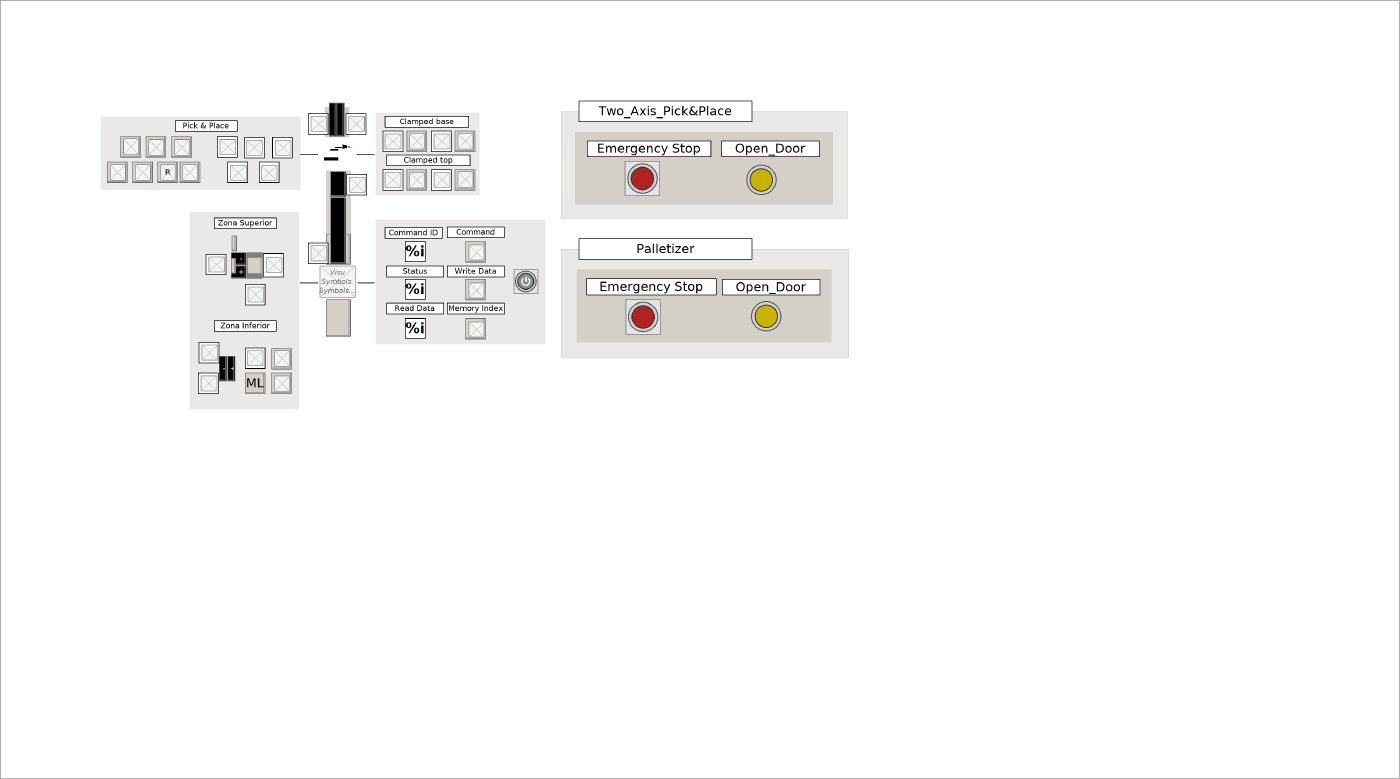
VISUALIZATION Linea_Produccion_Azul_2  // 2001x1114
    Rectangle (1846,508 153x409), angle 90
    Rectangle (827,144 248x30), "Two_Axis_Pick&Place"
    Rectangle (1855,498 103x368), angle 90
    PushSwitch (893,230 50x50), variable: GVL.Emergency_Stop_3, behaviour: TOGGLE, style: Switch-PushSwitch-Red
    Rectangle (839,201 177x23), "Emergency Stop"
    Lamp1 (1063,232 50x50), variable: NOT GVL.Safety_Door_1 OR NOT GVL.Safety_Door_2, style: Lamp-Lamp1-Yellow
    Rectangle (1031,201 140x23), "Open_Door"
    Rectangle (1846,703 155x411), angle 90
    Rectangle (827,341 248x30), "Palletizer"
    Rectangle (1614,447 104x364), angle 90
    PushSwitch (894,428 50x50), behaviour: TOGGLE, style: Switch-PushSwitch-Red
    Rectangle (838,398 186x24), "Emergency Stop"
    Lamp1 (1070,427 50x50), variable: NOT GVL.Safety_Door_3 OR NOT GVL.Safety_Door_4, style: Lamp-Lamp1-Yellow
    Rectangle (1032,399 140x23), "Open_Door"
    InvisibleInput (880,700 18x108)
    InvisibleInput (1316,220 49x41)
    Rectangle (1327,891 282x156), angle 90
    Rectangle (1569,733 118x148), angle 90
    Rectangle (1340,766 104x285), angle 90
    Button (466,334 35x44), colour toggle: GVL.Roller_Conveyor_2m_1, pressed state: GVL.Roller_Conveyor_2m_1
        OnMouseClick: toggle GVL.Roller_Conveyor_2m_1
    Rectangle (461,157 43x35), angle 90
    Group (456,196 53x49)
        InvisibleInput (0,0 53x49)
        RoundedRectangle (7,29 20x4), angle 107
        RoundedRectangle (16,17 11x2), angle 107
        RoundedRectangle (23,14 11x1), angle 180
        Polygon (33,10) (40,12) (40,14) (40,15) (33,17)
        Polygon (47,14) (47,14) (41,14) (41,14) (41,13)
    Rectangle (440,271 89x35), angle 90
    Group (455,378 55x50)
        InvisibleInput (0,0 55x50)
        Image (2,2 51x45), image: VisuSymbols.Symbols.Box
    Line (429,220) (454,220)
    Line (429,404) (454,404)
    Line (511,404) (535,404)
    Button (470,147 11x48), colour toggle: GVL.Belt_Conveyor_4m_6, pressed state: GVL.Belt_Conveyor_4m_6
        OnMouseClick: toggle GVL.Belt_Conveyor_4m_6
    Button (481,147 11x48), colour toggle: GVL.Belt_Conveyor_4m_7, pressed state: GVL.Belt_Conveyor_4m_7
        OnMouseClick: toggle GVL.Belt_Conveyor_4m_7
    Button (472,245 22x36), colour toggle: GVL.Belt_Conveyor_2m_15, pressed state: GVL.Belt_Conveyor_2m_15
        OnMouseClick: toggle GVL.Belt_Conveyor_2m_15
    Button (472,282 22x95), colour toggle: GVL.Belt_Conveyor_Inclined_1, pressed state: GVL.Belt_Conveyor_Inclined_1
        OnMouseClick: toggle GVL.Belt_Conveyor_Inclined_1
    Button (466,428 35x53), colour toggle: GVL.Roller_Conveyor_2m_2, pressed state: GVL.Roller_Conveyor_2m_2
        OnMouseClick: toggle GVL.Roller_Conveyor_2m_2
    Group (440,162 29x30), colour toggle: GVL.Diffuse_Sensor_12
        RoundedRectangle (0,0 29x30), colour toggle: GVL.Diffuse_Sensor_4
        Image (4,4 23x22), image: VisuSymbols.Symbols.RSS1
    Group (494,162 29x30), colour toggle: GVL.Diffuse_Sensor_13
        RoundedRectangle (0,0 29x30), colour toggle: GVL.Diffuse_Sensor_4
        Image (4,4 23x22), image: VisuSymbols.Symbols.RSS1
    Group (495,249 29x30), colour toggle: GVL.Diffuse_Sensor_14
        RoundedRectangle (0,0 29x30), colour toggle: GVL.Diffuse_Sensor_4
        Image (4,4 23x22), image: VisuSymbols.Symbols.RSS1
    Group (440,347 29x30), colour toggle: GVL.Diffuse_Sensor_22
        RoundedRectangle (0,0 29x30), colour toggle: GVL.Diffuse_Sensor_4
        Image (4,4 23x22), image: VisuSymbols.Symbols.RSS1
    Group (310,195 29x30), colour toggle: GVL.Two_Axis_Pick_Place_1_Detected
        RoundedRectangle (0,0 29x30), colour toggle: GVL.Two_Axis_Pick_Place_1_Detected
        Image (4,4 23x22), image: VisuSymbols.Symbols.RSS1
    Group (349,196 29x30), colour toggle: GVL.Two_Axis_Pick_Place_1_MovingX
        RoundedRectangle (0,0 29x30), colour toggle: GVL.Diffuse_Sensor_4
        Image (3,4 23x22), image: VisuSymbols.Symbols.DoubleArrow3
    Group (325,231 29x30), "G", colour toggle: GVL.Two_Axis_Pick_Place_1_Gripper_Rotating
        RoundedRectangle (0,0 29x30), colour toggle: GVL.Diffuse_Sensor_4
        Image (4,5 23x22), image: VisuSymbols.Symbols.ArrowRoundRightDown
    Group (389,196 29x30), colour toggle: GVL.Two_Axis_Pick_Place_1_MovingZ
        RoundedRectangle (0,0 29x30), colour toggle: GVL.Diffuse_Sensor_4
        Image (4,4 23x22), image: VisuSymbols.Symbols.DoubleArrow4
    Group (370,231 29x30), "R", colour toggle: GVL.Two_Axis_Pick_Place_1_Rotating
        RoundedRectangle (0,0 29x30), colour toggle: GVL.Diffuse_Sensor_4
        Image (3,5 23x22), image: VisuSymbols.Symbols.ArrowHalfLeftUp
    Rectangle (250,172 89x16), "Pick & Place"
    Group (547,187 29x30), colour toggle: NOT GVL.Right_Positioner_1_Clamped
        RoundedRectangle (0,0 29x30), colour toggle: GVL.Diffuse_Sensor_4
        Image (3,4 23x22), image: VisuSymbols.Symbols.DoubleArrow3
    Group (616,187 29x30), colour toggle: GVL.Right_Positioner_1_Limit
        RoundedRectangle (0,0 29x30), colour toggle: GVL.Diffuse_Sensor_4
        Image (4,4 23x22), image: VisuSymbols.Symbols.DoubleArrow4
    Rectangle (550,166 120x16), "Clamped base"
    Group (547,242 29x30), colour toggle: NOT GVL.Right_Positioner_2_Clamped
        RoundedRectangle (0,0 29x30), colour toggle: GVL.Diffuse_Sensor_4
        Image (3,4 23x22), image: VisuSymbols.Symbols.DoubleArrow3
    Group (616,242 29x30), colour toggle: GVL.Right_Positioner_2_Limit
        RoundedRectangle (0,0 29x30), colour toggle: GVL.Diffuse_Sensor_4
        Image (4,4 23x22), image: VisuSymbols.Symbols.DoubleArrow4
    Rectangle (552,221 120x16), "Clamped top"
    Line (510,220) (535,220)
    Button (330,361 22x18), "-", colour toggle: GVL.Palletizer_1_Belt_menos, pressed state: GVL.Palletizer_1_Belt_menos
        OnMouseClick: toggle GVL.Palletizer_1_Belt_menos
    Button (331,337 7x22), colour toggle: GVL.Palletizer_1_Turn, pressed state: GVL.Palletizer_1_Turn
        OnMouseClick: toggle GVL.Palletizer_1_Turn
    Button (353,361 22x36), colour toggle: GVL.Palletizer_1_Open_Plate, pressed state: GVL.Palletizer_1_Open_Plate
        OnMouseClick: toggle GVL.Palletizer_1_Open_Plate
    Button (353,391 22x7), colour toggle: GVL.Palletizer_1_Clamb, pressed state: GVL.Palletizer_1_Clamb
        OnMouseClick: toggle GVL.Palletizer_1_Clamb
    Group (350,406 29x30), colour toggle: GVL.Palletizer_1_Clamped
        RoundedRectangle (0,0 29x30), colour toggle: GVL.Diffuse_Sensor_4
        Image (4,4 23x22), image: VisuSymbols.Symbols.DoubleArrow4
    Group (376,362 29x34), colour toggle: GVL.Palletizer_1_Plate_Limit
        RoundedRectangle (0,0 29x34), colour toggle: GVL.Diffuse_Sensor_4
        Image (4,6 23x22), angle 45, image: VisuSymbols.Symbols.DoubleArrow1
    Button (330,380 22x18), "+", colour toggle: GVL.Palletizer_1_Belt_mas, pressed state: GVL.Palletizer_1_Belt_mas
        OnMouseClick: toggle GVL.Palletizer_1_Belt_mas
    Button (330,369 7x22), colour toggle: GVL.Palletizer_1_Push, pressed state: GVL.Palletizer_1_Push
        OnMouseClick: toggle GVL.Palletizer_1_Push
    Button (353,361 22x7), colour toggle: GVL.Palletizer_1_Clamb, pressed state: GVL.Palletizer_1_Clamb
        OnMouseClick: toggle GVL.Palletizer_1_Clamb
    Group (294,363 29x30), colour toggle: GVL.Palletizer_1_Pusher_Limit
        RoundedRectangle (0,0 29x30), colour toggle: GVL.Diffuse_Sensor_4
        Image (4,4 23x22), image: VisuSymbols.Symbols.ArrowBoldRight
    Button (325,509 11x36), "+", colour toggle: GVL.Palletizer_1_Chain_mas, pressed state: GVL.Palletizer_1_Belt_mas
        OnMouseClick: toggle GVL.Palletizer_1_Chain_mas
    Button (313,509 11x36), "-", colour toggle: GVL.Palletizer_1_Chain_menos, pressed state: GVL.Palletizer_1_Belt_menos
        OnMouseClick: toggle GVL.Palletizer_1_Chain_menos
    Group (284,489 29x30), colour toggle: GVL.Palletizer_1_Elevator_Back_Limit
        RoundedRectangle (0,0 29x30), colour toggle: GVL.Two_Axis_Pick_Place_1_Detected
        Image (4,4 23x22), image: VisuSymbols.Symbols.RSS1
    Group (283,533 29x30), colour toggle: GVL.Palletizer_1_Elevator_Front_Limit
        RoundedRectangle (0,0 29x30), colour toggle: GVL.Two_Axis_Pick_Place_1_Detected
        Image (4,4 23x22), image: VisuSymbols.Symbols.RSS1
    Group (350,497 29x30), colour toggle: GVL.Palletizer_1_Elevator_Moving
        RoundedRectangle (0,0 29x30), colour toggle: GVL.Diffuse_Sensor_4
        Image (3,4 23x22), image: VisuSymbols.Symbols.Wheel
    Button (350,533 29x30), "ML", colour toggle: GVL.Palletizer_1_Elevator_Move_Limit, pressed state: GVL.Palletizer_1_Open_Plate
        OnMouseClick: toggle GVL.Palletizer_1_Elevator_Move_Limit
    Group (388,498 29x30), colour toggle: GVL.Palletizer_1_Elevator_mas
        OnMouseClick: toggle GVL.Palletizer_1_Elevator_mas
        Button (0,0 29x30)
        Image (4,3 22x23), image: VisuSymbols.Symbols.ArrowBoldUp
    Group (388,533 29x30), colour toggle: GVL.Palletizer_1_Elevator_menos
        OnMouseClick: toggle GVL.Palletizer_1_Elevator_menos
        Button (0,0 29x30)
        Image (4,4 22x23), image: VisuSymbols.Symbols.ArrowBoldDown
    Rectangle (306,311 89x16), "Zona Superior"
    Rectangle (306,458 89x16), "Zona Inferior"
    Group (208,195 29x30), colour toggle: GVL.Two_Axis_Pick_Place_1X
        OnMouseClick: toggle GVL.Two_Axis_Pick_Place_1X
        Button (0,0 29x30)
        Image (4,4 22x23), image: VisuSymbols.Symbols.ArrowBoldRight
    Group (172,195 29x30), colour toggle: GVL.Two_Axis_Pick_Place_1_Grab
        OnMouseClick: toggle GVL.Two_Axis_Pick_Place_1_Grab
        Button (0,0 29x30)
        Image (4,3 22x23), image: VisuSymbols.Symbols.Download
    Group (257,231 29x30), colour toggle: GVL.Two_Axis_Pick_Place_1_Rotate_CCW
        OnMouseClick: toggle GVL.Two_Axis_Pick_Place_1_Rotate_CCW
        Button (0,0 29x30)
        Image (3,4 22x23), image: VisuSymbols.Symbols.ArrowHalfLeftUp
    Group (189,231 29x30), colour toggle: GVL.Two_Axis_Pick_Place_1_Gripper_CW
        OnMouseClick: toggle GVL.Two_Axis_Pick_Place_1_Gripper_CW
        Button (0,0 29x30)
        Image (4,4 22x23), image: VisuSymbols.Symbols.ArrowRoundRightDown
    Group (153,231 29x30), colour toggle: GVL.Two_Axis_Pick_Place_1_Gripper_CCW
        OnMouseClick: toggle GVL.Two_Axis_Pick_Place_1_Gripper_CCW
        Button (0,0 29x30)
        Image (4,4 22x23), image: VisuSymbols.Symbols.ArrowRoundLeftBottom
    Group (225,231 29x30), colour toggle: GVL.Two_Axis_Pick_Place_1_Rotare_CW
        OnMouseClick: toggle GVL.Two_Axis_Pick_Place_1_Rotare_CW
        Button (0,0 29x30)
        Image (4,4 22x23), "R", colour toggle: GVL.Two_Axis_Pick_Place_1_Rotate_CW, image: VisuSymbols.Symbols.ArrowHalfRightUp
            OnMouseClick: toggle GVL.Two_Axis_Pick_Place_1_Rotate_CW
    Group (245,195 29x30), colour toggle: GVL.Two_Axis_Pick_Place_1Z
        OnMouseClick: toggle GVL.Two_Axis_Pick_Place_1Z
        Button (0,0 29x30)
        Image (4,4 22x23), image: VisuSymbols.Symbols.ArrowBoldDown
    Group (581,187 29x30), colour toggle: GVL.Right_Positioner_1_Clamp
        OnMouseClick: toggle GVL.Right_Positioner_1_Clamp
        Button (0,0 29x30)
        Image (4,3 22x23), image: VisuSymbols.Symbols.DoubleArrow3
    Group (581,242 29x30), colour toggle: GVL.Right_Positioner_2_Clamp
        OnMouseClick: toggle GVL.Right_Positioner_2_Clamp
        Button (0,0 29x30)
        Image (4,4 22x23), image: VisuSymbols.Symbols.DoubleArrow3
    Group (650,242 29x30), colour toggle: GVL.Right_Positioner_2_Raise
        OnMouseClick: toggle GVL.Right_Positioner_2_Raise
        Button (0,0 29x30)
        Image (4,3 22x23), image: VisuSymbols.Symbols.ArrowBoldUp
    Group (650,187 29x30), colour toggle: GVL.Right_Positioner_1_Raise
        OnMouseClick: toggle GVL.Right_Positioner_1_Raise
        Button (0,0 29x30)
        Image (4,3 22x23), image: VisuSymbols.Symbols.ArrowBoldUp
    Rectangle (1569,792 178x242), angle 90
    Rectangle (579,345 29x29), "%i", text variable: GVL.RFID_Reader_1_Command_ID
        p4168582468: GVL.RFID_Reader_1_Command_ID
    Rectangle (550,325 82x16), "Command ID"
    Rectangle (552,380 82x16), "Status"
    Rectangle (552,433 82x16), "Read Data"
    Rectangle (579,399 29x29), "%i", text variable: GVL.RFID_Reader_1_Status
        p4168582468: GVL.RFID_Reader_1_Status
    Rectangle (579,455 29x29), "%i", text variable: GVL.RFID_Reader_1_Read_Data
        p4168582468: GVL.RFID_Reader_1_Read_Data
    PowerSwitch (734,385 35x35), variable: GVL.RFID_Reader_1_Ejecute_Comm, behaviour: TOGGLE, style: Switch-PowerSwitch-Gray
    Rectangle (639,324 82x16), "Command"
    Rectangle (639,380 82x16), "Write Data"
    Rectangle (639,433 82x16), "Memory Index"
    Group (665,345 29x30)
        OnMouseClick: write GVL.RFID_Reader_1_Command_ID via VisuDialogs.Numpad, min 0, max 100, format %i
        Button (0,0 29x30), text variable: GVL.RFID_Reader_1_Command
            OnMouseClick: write GVL.RFID_Reader_4_Command_ID via VisuDialogs.Numpad, min 0, max 100, format %i
        Image (5,5 22x22), image: VisuSymbols.Symbols.Edit
    Group (665,399 29x30)
        OnMouseClick: write GVL.RFID_Reader_1_Write_Data via VisuDialogs.Numpad, min 0, max 100, format %i
        Button (0,0 29x30), text variable: GVL.RFID_Reader_1_Command
            OnMouseClick: write GVL.RFID_Reader_4_Command_ID via VisuDialogs.Numpad, min 0, max 100, format %i
        Image (5,5 22x22), image: VisuSymbols.Symbols.Edit
    Group (665,455 29x30)
        OnMouseClick: write GVL.RFID_Reader_1_Memory_Index via VisuDialogs.Numpad, min 0, max 100, format %i
        Button (0,0 29x30), text variable: GVL.RFID_Reader_1_Command
            OnMouseClick: write GVL.RFID_Reader_4_Command_ID via VisuDialogs.Numpad, min 0, max 100, format %i
        Image (5,5 22x22), image: VisuSymbols.Symbols.Edit
END_VISUALIZATION

(* stored: Version 1.1.0.1, ProductVersion 3.1.4024.12
   Visu Linea_Produccion_Azul_2: Id {b2c0885e-ed2a-41d4-be15-ceffd1454d2b} *)
